Staubli VAL3: loadmaster9.pgx

program loadmaster9(string x_sMasterFile9 (dimensions=1))
begin
  if master:libLoad(x_sMasterFile9)<0
    popUpMsg("nO ok")
  endIf
  frmaster[9].trsf=master:tTool.trsf
  //取个数
  nsize[9]=size(master:ptRoutingPath)
  //存个数
  resize(pdemo9,1,nsize[9])
  //保存程序
  master:libSave()
end
